(* IEC 61131-3 sources: ATCMcontrol_Engineering/src/TargetBase/Libs/Datalogger, 4 files *)

(* ---- Datalog_eject.st ---- *)
(*[[
    UserHelpURL= "ATCMfile:Datalog_eject.HTML",
]]*)
FUNCTION Datalog_eject : UINT
VAR_INPUT
        index : UINT;
END_VAR
	INLINE {STDLIB(Datalog_eject)}
END_FUNCTION

(* ---- Datalog_get.st ---- *)
(*[[
    UserHelpURL= "ATCMfile:Datalog_get.HTML",
]]*)
FUNCTION Datalog_get : UINT
VAR_INPUT
        label : STRING;
        value : REAL;
END_VAR
	INLINE {STDLIB(Datalog_get)}
END_FUNCTION

(* ---- Datalog_start.st ---- *)
(*[[
    UserHelpURL= "ATCMfile:Datalog_start.HTML",
]]*)
FUNCTION Datalog_start : INT
VAR_INPUT
        buffer_lenght : UDINT;
        buffer_number : UINT;
        index : UINT;
END_VAR
	INLINE {STDLIB(Datalog_start)}
END_FUNCTION

(* ---- Datalog_stop.st ---- *)
(*[[
    UserHelpURL= "ATCMfile:Datalog_stop.HTML",
]]*)
FUNCTION Datalog_stop : UINT
	INLINE {STDLIB(Datalog_stop)}
END_FUNCTION
